{attribute 'linkalways'} 
{attribute 'no_explicit_call' := 'This FB is a CLASS and must be accessed using methods or properties'}
{attribute 'enable_dynamic_creation'}
FUNCTION_BLOCK FINAL LOG_LREAL EXTENDS Node
VAR
	in : _LREAL(0.0);
	out : _LREAL(0.0);
END_VAR

METHOD PUBLIC Clone : I_Node
VAR
	pNode : POINTER TO LOG_LREAL;
END_VAR
pNode := __NEW(LOG_LREAL);
Clone := pNode^;
END_METHOD

METHOD FB_init : BOOL
VAR_INPUT
	bInitRetains : BOOL; // if TRUE, the retain variables are initialized (warm start / cold start)
	bInCopyCode : BOOL;  // if TRUE, the instance afterwards gets moved into the copy code (online change)
END_VAR
AddInput('in',THIS^.in);
AddOutput('out', THIS^.out);
END_METHOD

METHOD PROTECTED OnExecute
VAR
END_VAR
out.Value := LOG(in.Value);
END_METHOD

END_FUNCTION_BLOCK

(* stored: Version 1.1.0.1, ProductVersion 3.1.4024.15
   POU LOG_LREAL: Id {6e946d79-a0b9-4ecf-ae03-f0e18f12c803}, SpecialFunc None
   Folder Constructor: Id {dbf9936a-4cab-4390-a32c-2873d3414851}
   Method Clone: Id {87c8bb96-652b-4331-a1e1-794dd9f8a258}
   Method FB_init: Id {3f65ddd3-f3a3-41fc-95ba-b01a8164848a}
   Method OnExecute: Id {2a089367-bb52-4659-af7a-be0bcb8a59a3} *)
